// TIA Portal V15.1 export
// export: Created 2022-09-01T22:37:49.1492764Z, ExportSetting WithDefaults, WithReadOnly, DisplayName Totally Integrated Automation Portal, DisplayVersion V15.1 Update 5, DisplayName TIA Portal Openness, DisplayVersion V15.1 Update 5, DisplayName STEP 7 Professional, DisplayVersion V15.1 Update 5, DisplayName WinCC Advanced, DisplayVersion V15.1 Update 5
FUNCTION "Teste_XML" : Void   // FC2, LAD
{ S7_Optimized_Access := 'TRUE' }
VERSION : 0.1
// stored: AutoNumber true, CodeModifiedDate 2022-09-01T22:36:45.9032848Z, CompileDate 2022-09-01T22:36:47.5161826Z, CreationDate 2022-09-01T22:29:47.8545045Z, HandleErrorsWithinBlock false, InterfaceModifiedDate 2022-09-01T22:32:46.4008877Z, IsConsistent true, IsIECCheckEnabled false, IsKnowHowProtected false, IsWriteProtected false, LibraryConformanceStatus The object is library-conformant., ModifiedDate 2022-09-01T22:36:45.9032848Z, ParameterModified 2022-09-01T22:32:46.4008877Z, PLCSimAdvancedSupport true, SetENOAutomatically False, StructureModified 2022-09-01T22:32:46.4008877Z, UDAEnableTagReadback false
   VAR_INPUT
      Tag1 : Bool;
      Tag2 : Bool;
   END_VAR
   VAR_OUTPUT
      Tag4 : Bool;
   END_VAR
   VAR_IN_OUT
      Tag3 : Bool;
   END_VAR
BEGIN

REGION Network 1: Teste
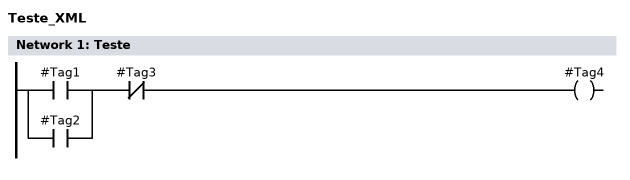
   RUNG wire#powerrail
      Contact( #Tag1 )
      wire#w1
      I_Contact( #Tag3 )
      Coil( #Tag4 )
   END_RUNG
   RUNG wire#powerrail
      Contact( #Tag2 )
   END_RUNG wire#w1
   // the same network as SCL:
   #Tag4 := (#Tag1 OR #Tag2) AND NOT #Tag3;
END_REGION
END_FUNCTION
